{attribute 'qualified_only'}
VAR_GLOBAL
	NumericValue_10ms : INT;
	NumericValue_100ms : INT;
	NumericValue_1000ms : INT;
	Numericvalue_Constant : INT := 12245;
END_VAR

(* stored: Version 1.1.0.1, ProductVersion 3.1.4024.12
   GVL GVL_Subscription: Id {ec6673ea-66c8-4cb2-a1d4-20a14c59190b} *)
